// TIA Portal V20 export
DATA_BLOCK "STATION"   // DB49
{ S7_Optimized_Access := 'TRUE' }
VERSION : 0.1
// stored: AutoNumber true, DBAccessibleFromOPCUA true, DBAccessibleFromWebserver true, IsOnlyStoredInLoadMemory false, IsRetainMemResEnabled false, IsWriteProtectedInAS false, MemoryReserve 100
   VAR RETAIN
      Count : UInt := 32;
      Station : Array["STATION_MIN".."STATION_MAX"] of "LGR_Station_Para";
   END_VAR
BEGIN
END_DATA_BLOCK
